PROGRAM MAIN
VAR
END_VAR

END_PROGRAM

(* stored: Version 1.1.0.1
   POU MAIN: Id {2ccece19-8542-4c6e-8089-770971141e6d} *)
